FUNCTION_BLOCK Drive1 EXTENDS DriveBase
VAR_INPUT
END_VAR
VAR_OUTPUT
END_VAR
VAR
END_VAR

{error 'Add method implementation or delete method to use base implementation'}
METHOD Disable : BOOL
END_METHOD

{error 'Add method implementation or delete method to use base implementation'}
METHOD Enable : BOOL
END_METHOD

END_FUNCTION_BLOCK

(* stored: Version 1.1.0.1
   POU Drive1: Id {3555369e-3e13-48b4-b985-4b5677e918ce}, SpecialFunc None
   Method Disable: Id {fc7ec26f-845d-492e-8ed0-6648374057c1}
   Method Enable: Id {5a8a7da1-54e0-4243-8466-b125c2019fb8} *)
